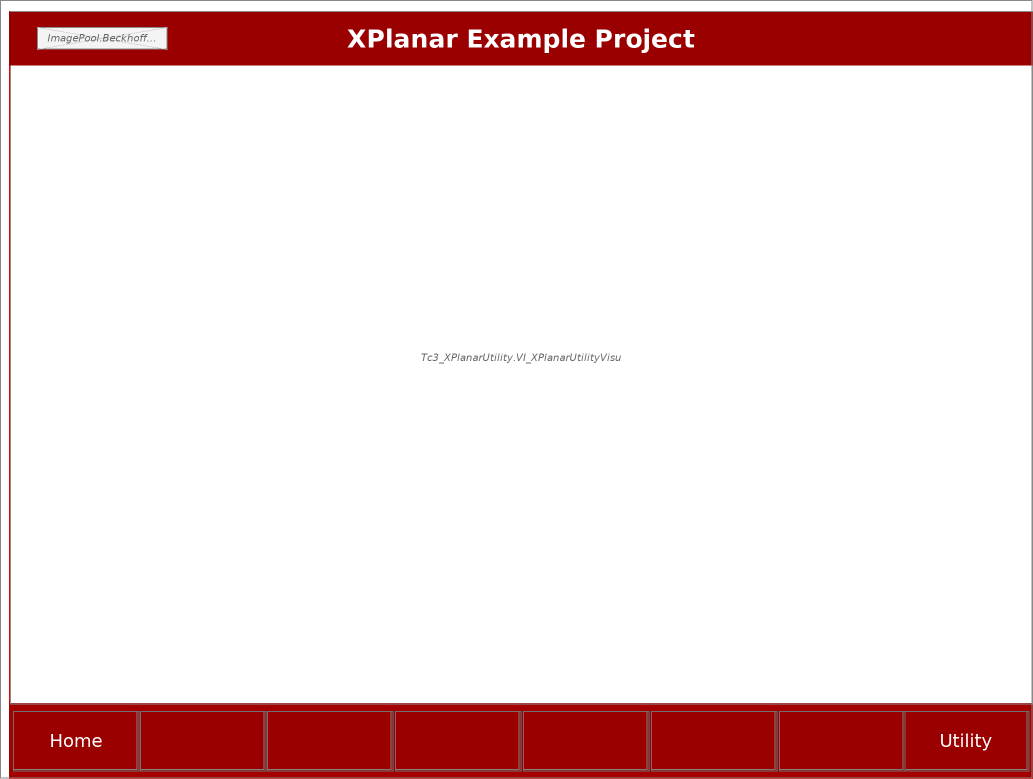
VISUALIZATION UtilityPage  // 1033x779
    Rectangle (9,11 1024x768)
    Rectangle (9,703 1024x75)
    Button (13,711 126x60), "Home"
        OnMouseDown: change screen: Visualization
    Button (140,711 126x60)
    Button (903,711 126x60), "Utility"
        OnMouseUp: change screen: UtilityPage
    Button (395,711 126x60)
    Button (523,711 126x60)
    Button (651,711 126x60)
    Button (779,711 126x60)
    Button (267,711 126x60)
    Frame (10,11 1023x693)
        shows Tc3_XPlanarUtility.VI_XPlanarUtilityVisu()
    Group (9,12 1024x53)
        Image (18,11 130x22), image: ImagePool.Beckhoff_white
        Rectangle (0,0 1024x53), "XPlanar Example Project"
        Image (28,15 130x22), image: ImagePool.Beckhoff_white
END_VISUALIZATION

(* stored: Version 1.1.0.1
   Visu UtilityPage: Id {7517170f-a536-4135-b17a-e3864af6a176} *)
